FUNCTION_BLOCK FB_Math
VAR_INPUT
END_VAR
VAR_OUTPUT
END_VAR
VAR
	{attribute 'OPC.UA.DA':='1'}
	nNumberOfCallsMMul : INT;
	{attribute 'OPC.UA.DA':='1'}
	nNumberOfCallsMAdd : INT;
	{attribute 'OPC.UA.DA':='1'}
	nNumberOfCallsMRpm : INT;
END_VAR

{attribute 'TcRpcEnable':='1'}
METHOD M_Add : DINT
VAR_INPUT
	a : INT;
	b : INT;
END_VAR
M_Add := a + b;
nNumberOfCallsMAdd := nNumberOfCallsMAdd + 1;
END_METHOD

{attribute 'TcRpcEnable':='1'}
METHOD M_Mul : DINT
VAR_INPUT
	a : INT;
	b : INT;
END_VAR
M_Mul := a * b;
nNumberOfCallsMMul := nNumberOfCallsMMul + 1;
END_METHOD

{attribute 'TcRpcEnable':='1'}
METHOD M_Rpm : DINT
VAR_INPUT
	motorSpeed : DINT;
	gearboxRatio : DINT;
END_VAR
M_Rpm := motorSpeed/gearboxRatio;
nNumberOfCallsMRpm := nNumberOfCallsMRpm + 1;
END_METHOD

END_FUNCTION_BLOCK

(* stored: Version 1.1.0.1, ProductVersion 3.1.4024.11
   POU FB_Math: Id {d21c0b8e-6469-45a1-ba1e-9bee226b3d60}, SpecialFunc None
   Method M_Add: Id {1e1b49ec-5f56-4257-ba09-e8dd62db2c6f}
   Method M_Mul: Id {ce515e7e-be6c-41f1-9c46-1955d83b401d}
   Method M_Rpm: Id {63435d25-8cf9-4de1-b56f-5b99f79ae5e2} *)
